PROGRAM MAIN
VAR
	sampleTime: REAL := 0.5;
	state: INT	:=	0;	
	start: BOOL	:=	FALSE;
	operationModeWrite: SINT	:=	10;	
	
	{attribute 'TcNcAxis' := '[0]:=Axis 1;[1]:=Axis 2;[2]:=Axis 3'} 
    // Using an axis in an array.
    setAxis     : ARRAY [0..2] OF AXIS_REF;
	
	opertionModeRead: SINT;
	
	fbCoERead: FB_CoERead;
	
	MotorEnable: BOOL:=FALSE;
	
	mcReset: MC_Reset;
	mcPower: MC_Power;
	
////////
	
	operitonModeCh: WORD;
	subIndex: BYTE;	
	axisSelect: (xAxis, yAxis, zAxis, xyAxis, allAxis);	
	fbCoEWrite: FB_CoEWrite;	
	//torque : FB_TorqueInput;
	
END_VAR
VAR_INPUT
	dummy : INT ;
END_VAR

CASE state OF
	//Axis Selection
0:
	IF start THEN
		
		IF axisSelect = xAxis THEN
			operitonModeCh := 16#6060;
			subIndex := 0;
			MotorEnable:=TRUE;
			dummy := 0;	
		ELSIF axisSelect = yAxis THEN	
			operitonModeCh := 16#6860;		
			subIndex := 0;
			MotorEnable:=TRUE;	
			dummy := 1;	
		ELSIF axisSelect = zAxis THEN	
			operitonModeCh := 16#6860;
			MotorEnable:=TRUE;	
			dummy := 2;
			subIndex := 0;
			
		ELSIF axisSelect = xyAxis THEN	
			operitonModeCh := 16#6860;
			MotorEnable:=TRUE;	
			dummy := 3;
			subIndex := 0;
		END_IF
		
		state:=190;
		start:=FALSE;		
	END_IF

190:
	mcReset(
	Axis:=setAxis[dummy] , 
	Execute:=TRUE , 
	 );
	IF NOT mcReset.Busy AND mcReset.Done THEN		
		mcReset(Axis:=setAxis[dummy], Execute:=FALSE);		
		state:=200;
	END_IF
	
	//Mod of operation
200:


	fbCoEWrite(
		Axis:= setAxis[dummy], 
		NetId:='', 
		Index:= operitonModeCh, 
		SubIndex:=subIndex,
		pSrcBuf:= ADR(operationModeWrite), 
		BufLen:= SIZEOF(operationModeWrite), 
		Execute:=TRUE , 		
		CompleteAccess:=TRUE , 
		 );
		
	IF NOT fbCoEWrite.Busy THEN
		fbCoEWrite(
		Axis:= setAxis[dummy], 
		NetId:='', 
		Index:= operitonModeCh, 
		SubIndex:=subIndex, 
		pSrcBuf:= ADR(operationModeWrite), 
		BufLen:= SIZEOF(operationModeWrite), 
		Execute:=FALSE , 		
		CompleteAccess:=TRUE , 
		 );
		
		fbCoERead(
			Axis:=setAxis[dummy] , 
			NetId:= '', 
			Index:= operitonModeCh,
			SubIndex:= subIndex,
			pDstBuf:= ADR(opertionModeRead), 
			BufLen:= SIZEOF(opertionModeRead), 
			Execute:= TRUE, 			
			CompleteAccess:=TRUE , 
			 );
			
			IF opertionModeRead = operationModeWrite AND NOT fbCoERead.Busy THEN
			
				fbCoeRead(Axis:=setAxis[dummy],Execute:=FALSE );
				IF NOT fbCoERead.Execute THEN
					state:=210;
				END_IF
			END_IF
	END_IF
	
	//power enable
	//motor enable
210:
	mcReset(
	Axis:=setAxis[dummy] , 
	Execute:=TRUE , 
	 );
	IF NOT mcReset.Busy AND mcReset.Done THEN		
		mcReset(Axis:=setAxis[dummy], Execute:=FALSE);		
		state:=220;
	END_IF
	
	220:
	
	mcPower(
	Axis:=setAxis[dummy] , 
	Enable:= MotorEnable , 
	Enable_Positive:= MotorEnable, 
	Enable_Negative:= MotorEnable, 
 );
	IF (mcPower.Status AND MotorEnable) OR (NOT mcPower.Status AND NOT MotorEnable) THEN 

		state:=230;
	END_IF
	

230:

// 	torque(torqueInput:=20, duration:=2);
//	IF torque.busy = FALSE THEN
//		state := 232;
//	END_IF

 
232:
  
// velocityInput();
// IF NOT velocityInput.busy THEN
//	 state := 240;
// END_IF
 
240 :
 mcReset(
	Axis:=setAxis[dummy] , 
	Execute:=TRUE , 
	 );
	IF NOT mcReset.Busy AND mcReset.Done THEN		
		mcReset(Axis:=setAxis[dummy], Execute:=FALSE);		
		state:=250;
	END_IF
 
	250:
 	MotorEnable := FALSE;
 	mcPower(
	Axis:=setAxis[dummy] , 
	Enable:= MotorEnable , 
	Enable_Positive:= MotorEnable, 
	Enable_Negative:= MotorEnable, 
 );
	IF (mcPower.Status AND MotorEnable) OR (NOT mcPower.Status AND NOT MotorEnable) THEN 
		state:=260;
	END_IF
	//Motor disable
260:
 	

	state := 0;

END_CASE

END_PROGRAM

(* stored: Version 1.1.0.1, ProductVersion 3.1.4024.9
   POU MAIN: Id {d4c23686-4223-4849-8fc3-1f69218d516d}, SpecialFunc None *)
